(* Logix 5000 project; controller RN21_Architecture 1769-L16ER-BB1B rev 35.11; software revision 35.00; part 2 of 9 *)

ADD_ON_INSTRUCTION AOI_LOGIN_Arch   (* revision 1.0 *)
VAR_INPUT
   FBI_DataLogTrig : BOOL; {required}   // Trigger Bit for Data Log Generation
END_VAR
VAR_IN_OUT
   FBO_TriggerBit : BOOL; {required}   // Server Trigger Bit
   FBIO_Src : UDT_Login; {required}   // Source UDT Data
   FBIO_Ser : UDT_Login; {required}   // Server UDT Data
END_VAR
VAR_INPUT
   FBI_PLCServerCommFailed : BOOL; {access None, required}   // PLC to Server Communication Fail Timer Done
END_VAR
VAR_IN_OUT
   FBIO_SerUniqueNum : DINT; {required}   // Server Unique Number(Server UID)
   FBIO_SrcUniqueNum : DINT; {required}   // Source Unique Number (PLC UID)
END_VAR
VAR
   FBL_Buff : UDT_Login[100]; {access None}   // Buffer UDT Data
   FBL_Sec : UDT_Login; {access None}   // Secondary UDT Data
   FBL_IndexStore : DINT; {access None}   // Index Store Value
   FBL_Bit4 : BOOL; {access None}   // Primary Movement Completed
   FBL_TMR2 : TIMER := (PRE := 50, ACC := 1); {access None}   // Source UID Reset Delay
   FBL_Bit1 : BOOL; {access None}   // Source UID Reset
   FBL_Bit2 : BOOL; {access None}   // Source UID Less than Server UID
   FBL_Bit6 : BOOL; {access None}   // Data Moving From Secondary to Server
   FBL_TMR3 : TIMER := (PRE := 5000, ACC := 5); {access None}   // Load Movement Delay
   FBL_Bit5 : BOOL; {access None}   // Data Load From Buffer to Secondary Flag
   FBL_IndexLoad : DINT; {access None}   // Index Load Value
   FBL_Bit3 : BOOL; {access None}   // Secondary Movement Completed
   FBL_TMR1 : TIMER := (PRE := 5000); {access None}   // Server UID Movement Delay
   FBL_PrimUniqueNum : DINT; {access None}   // Primary Unique Number (PLC UID)
   FBL_BuffUniqueNum : DINT[100]; {access None}   // Buffer Unique Number (PLC UID)
   FBL_SecUniqueNum : DINT; {access None}   // Secondary Unique Number (PLC UID)
   FBL_Prim : UDT_Login; {access None}   // Primary UDT Data
   FBL_ONS : DINT; {access None}   // Common ONS DINT
   TMRDlyDatalogTrig : TIMER := (PRE := 1); {access None}
END_VAR

ROUTINE Logic   (* ladder *)
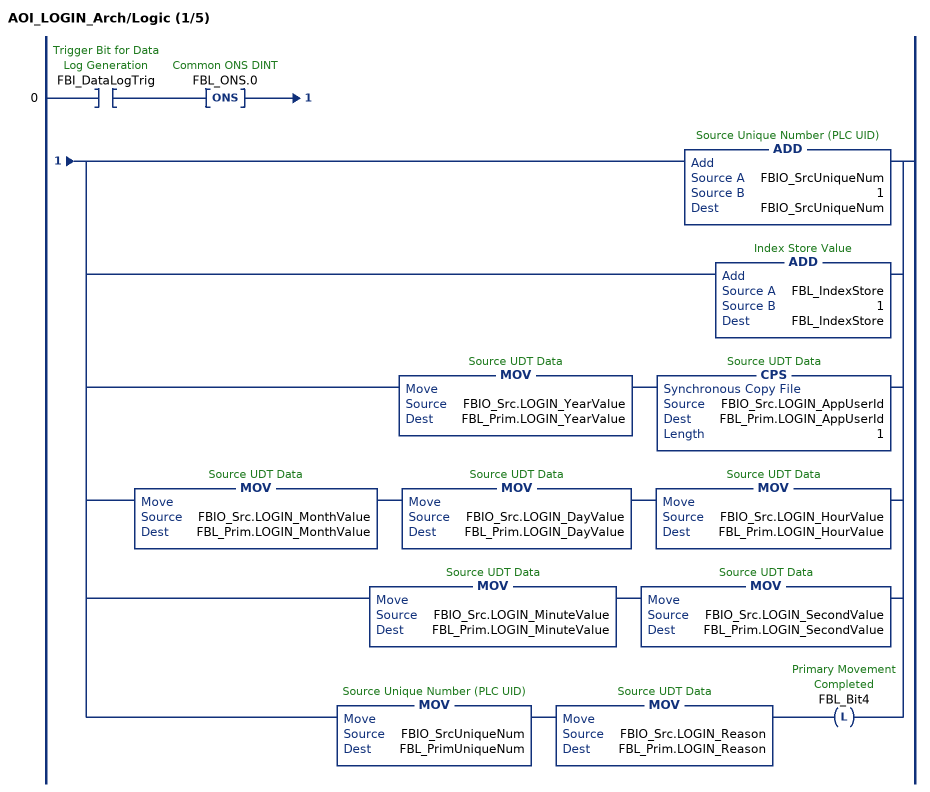
   0: XIC(FBI_DataLogTrig)ONS(FBL_ONS.0)[ADD(FBIO_SrcUniqueNum,1,FBIO_SrcUniqueNum) ,ADD(FBL_IndexStore,1,FBL_IndexStore) ,MOV(FBIO_Src.LOGIN_YearValue,FBL_Prim.LOGIN_YearValue) CPS(FBIO_Src.LOGIN_AppUserId,FBL_Prim.LOGIN_AppUserId,1) ,MOV(FBIO_Src.LOGIN_MonthValue,FBL_Prim.LOGIN_MonthValue) MOV(FBIO_Src.LOGIN_DayValue,FBL_Prim.LOGIN_DayValue) MOV(FBIO_Src.LOGIN_HourValue,FBL_Prim.LOGIN_HourValue) ,MOV(FBIO_Src.LOGIN_MinuteValue,FBL_Prim.LOGIN_MinuteValue) MOV(FBIO_Src.LOGIN_SecondValue,FBL_Prim.LOGIN_SecondValue) ,MOV(FBIO_SrcUniqueNum,FBL_PrimUniqueNum) MOV(FBIO_Src.LOGIN_Reason,FBL_Prim.LOGIN_Reason) OTL(FBL_Bit4) ];
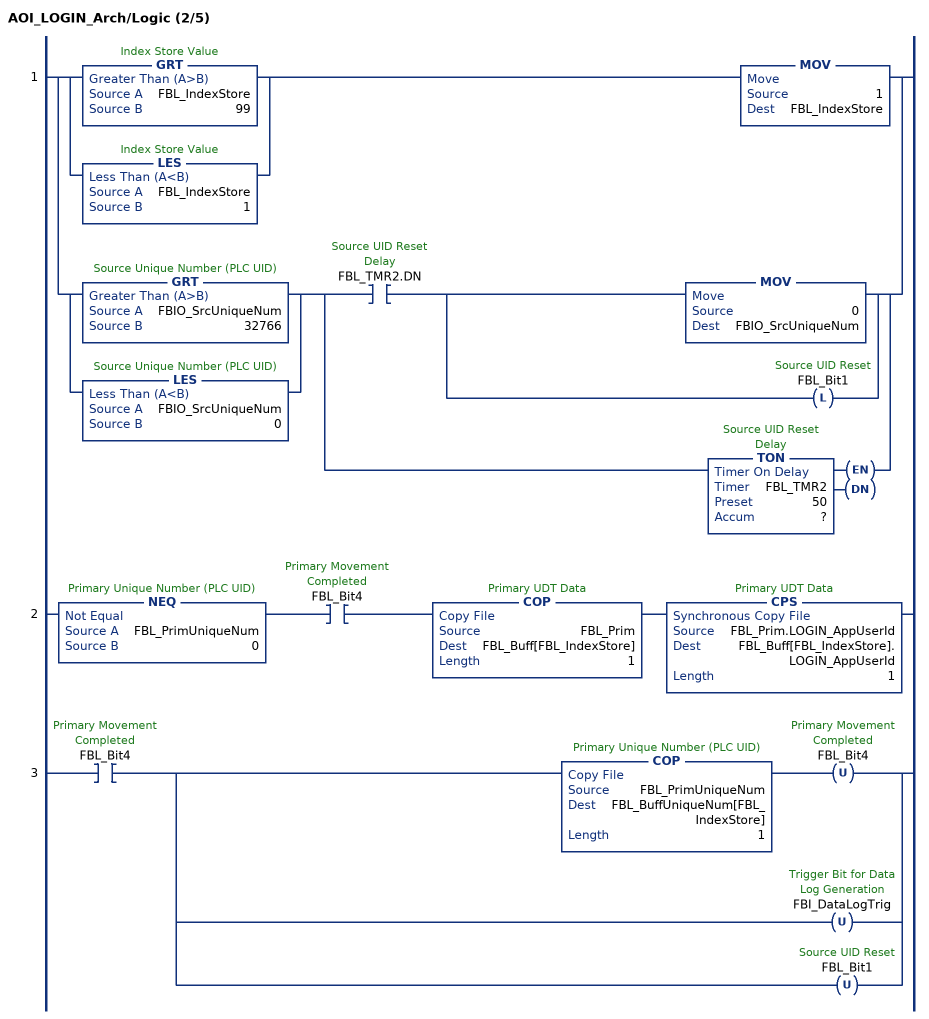
   1: [[GRT(FBL_IndexStore,99) ,LES(FBL_IndexStore,1) ] MOV(1,FBL_IndexStore) ,[GRT(FBIO_SrcUniqueNum,32766) ,LES(FBIO_SrcUniqueNum,0) ] [XIC(FBL_TMR2.DN) [MOV(0,FBIO_SrcUniqueNum) ,OTL(FBL_Bit1) ] ,TON(FBL_TMR2,?,?) ] ];
   2: NEQ(FBL_PrimUniqueNum,0)XIC(FBL_Bit4)COP(FBL_Prim,FBL_Buff[FBL_IndexStore],1)CPS(FBL_Prim.LOGIN_AppUserId,FBL_Buff[FBL_IndexStore].LOGIN_AppUserId,1);
   3: XIC(FBL_Bit4)[COP(FBL_PrimUniqueNum,FBL_BuffUniqueNum[FBL_IndexStore],1) OTU(FBL_Bit4) ,OTU(FBI_DataLogTrig) ,OTU(FBL_Bit1) ];
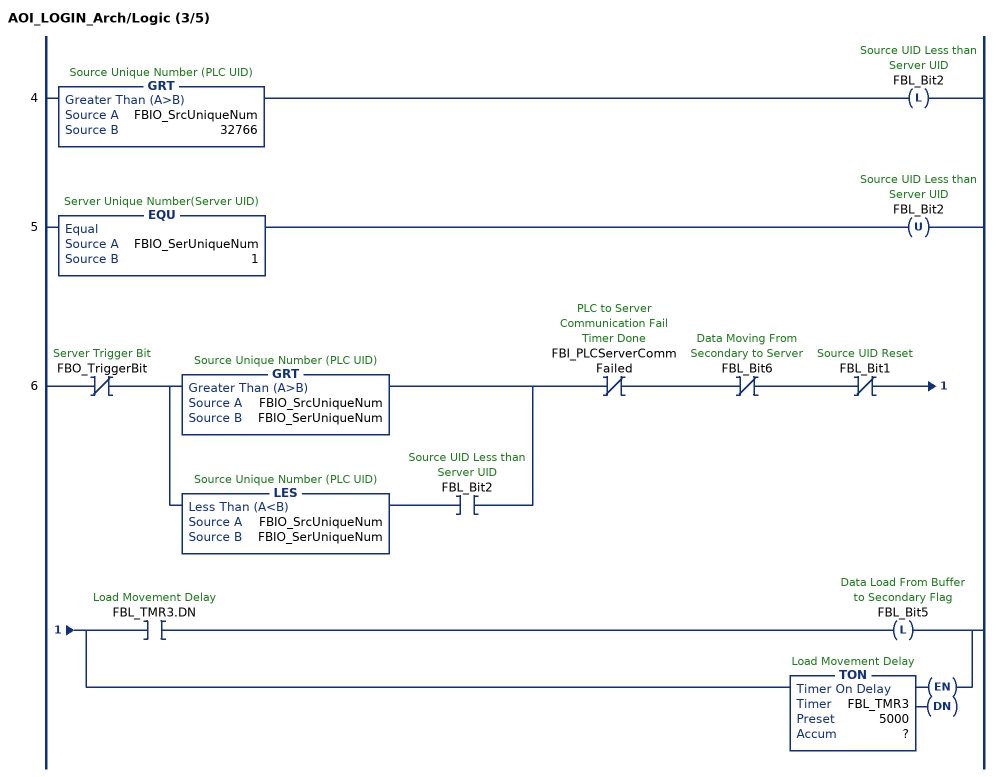
   4: GRT(FBIO_SrcUniqueNum,32766)OTL(FBL_Bit2);
   5: EQU(FBIO_SerUniqueNum,1)OTU(FBL_Bit2);
   6: XIO(FBO_TriggerBit)[GRT(FBIO_SrcUniqueNum,FBIO_SerUniqueNum) ,LES(FBIO_SrcUniqueNum,FBIO_SerUniqueNum) XIC(FBL_Bit2) ]XIO(FBI_PLCServerCommFailed)XIO(FBL_Bit6)XIO(FBL_Bit1)[XIC(FBL_TMR3.DN) OTL(FBL_Bit5) ,TON(FBL_TMR3,?,?) ];
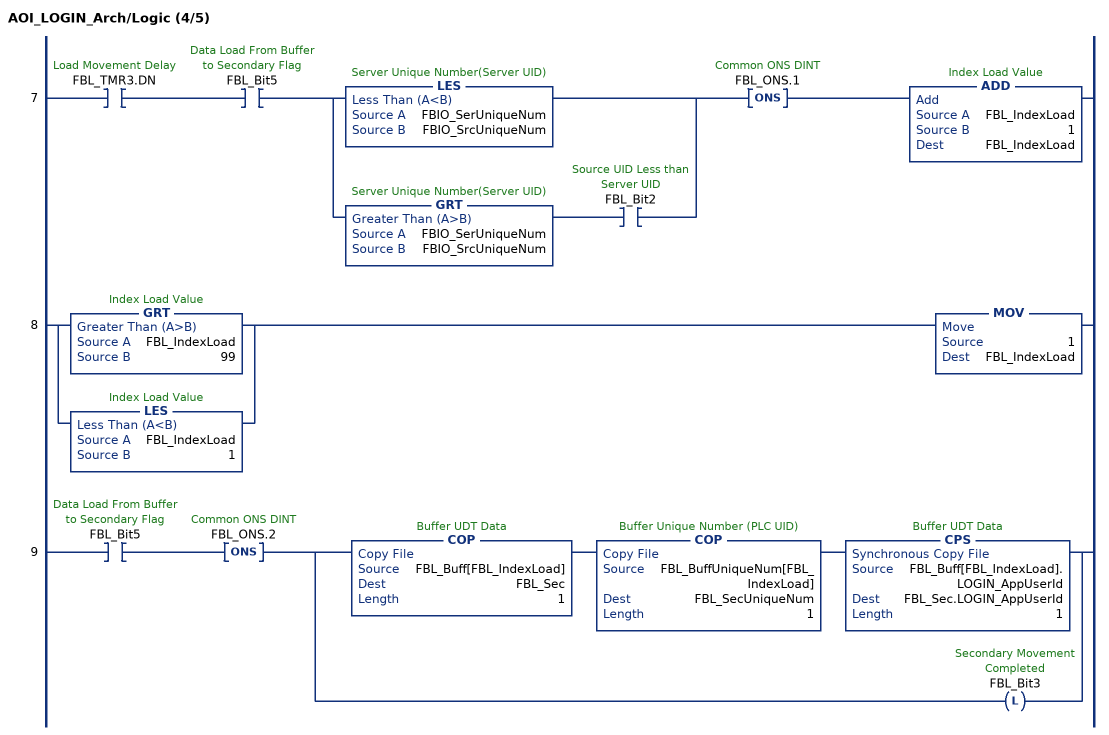
   7: XIC(FBL_TMR3.DN)XIC(FBL_Bit5)[LES(FBIO_SerUniqueNum,FBIO_SrcUniqueNum) ,GRT(FBIO_SerUniqueNum,FBIO_SrcUniqueNum) XIC(FBL_Bit2) ]ONS(FBL_ONS.1)ADD(FBL_IndexLoad,1,FBL_IndexLoad);
   8: [GRT(FBL_IndexLoad,99) ,LES(FBL_IndexLoad,1) ]MOV(1,FBL_IndexLoad);
   9: XIC(FBL_Bit5)ONS(FBL_ONS.2)[COP(FBL_Buff[FBL_IndexLoad],FBL_Sec,1) COP(FBL_BuffUniqueNum[FBL_IndexLoad],FBL_SecUniqueNum,1) CPS(FBL_Buff[FBL_IndexLoad].LOGIN_AppUserId,FBL_Sec.LOGIN_AppUserId,1) ,OTL(FBL_Bit3) ];
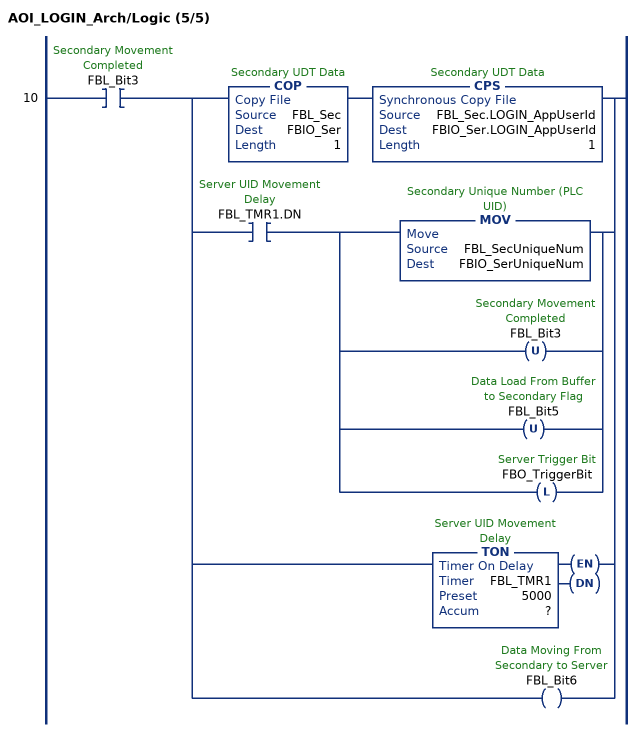
   10: XIC(FBL_Bit3)[COP(FBL_Sec,FBIO_Ser,1) CPS(FBL_Sec.LOGIN_AppUserId,FBIO_Ser.LOGIN_AppUserId,1) ,XIC(FBL_TMR1.DN) [MOV(FBL_SecUniqueNum,FBIO_SerUniqueNum) ,OTU(FBL_Bit3) ,OTU(FBL_Bit5) ,OTL(FBO_TriggerBit) ] ,TON(FBL_TMR1,?,?) ,OTE(FBL_Bit6) ];
END_ROUTINE
END_ADD_ON_INSTRUCTION

ADD_ON_INSTRUCTION AOI_PDL_Arch   (* revision 1.0 *)
VAR_INPUT
   FBI_DataLogTrig : BOOL; {required}   // Trigger Bit for Data Log Generation
END_VAR
VAR_IN_OUT
   FBO_TriggerBit : BOOL; {required}   // Server Trigger Bit
   FBIO_Src : UDT_Process; {required}   // Source UDT Data
   FBIO_Ser : UDT_Process; {required}   // Server UDT Data
END_VAR
VAR_INPUT
   FBI_PLCServerCommFailed : BOOL; {access None, required}   // PLC to Server Communication Fail Timer Done
END_VAR
VAR_IN_OUT
   FBIO_SerUniqueNum : DINT; {required}   // Server Unique Number(Server UID)
   FBIO_SrcUniqueNum : DINT; {required}   // Source Unique Number (PLC UID)
END_VAR
VAR
   FBL_Prim : UDT_Process; {access None}   // Primary UDT Data
   FBL_Buff : UDT_Process[100]; {access None}   // Buffer UDT Data
   FBL_Sec : UDT_Process; {access None}   // Secondary UDT Data
   FBL_IndexStore : DINT; {access None}   // Index Store Value
   FBL_Bit4 : BOOL; {access None}   // Primary Movement Completed
   FBL_TMR2 : TIMER := (PRE := 1, ACC := 1); {access None}   // Source UID Reset Delay
   FBL_Bit1 : BOOL; {access None}   // Source UID Reset
   FBL_Bit2 : BOOL; {access None}   // Source UID Less than Server UID
   FBL_Bit6 : BOOL; {access None}   // Data Moving From Secondary to Server
   FBL_TMR3 : TIMER := (PRE := 5000, ACC := 5); {access None}   // Load Movement Delay
   FBL_Bit5 : BOOL; {access None}   // Data Load From Buffer to Secondary Flag
   FBL_IndexLoad : DINT; {access None}   // Index Load Value
   FBL_Bit3 : BOOL; {access None}   // Secondary Movement Completed
   FBL_TMR1 : TIMER := (PRE := 5000); {access None}   // Server UID Movement Delay
   FBL_PrimUniqueNum : DINT; {access None}   // Primary Unique Number (PLC UID)
   FBL_BuffUniqueNum : DINT[100]; {access None}   // Buffer Unique Number (PLC UID)
   FBL_SecUniqueNum : DINT; {access None}   // Secondary Unique Number (PLC UID)
   FBL_ONS : DINT; {access None}   // Common ONS DINT
END_VAR

ROUTINE Logic   (* ladder *)
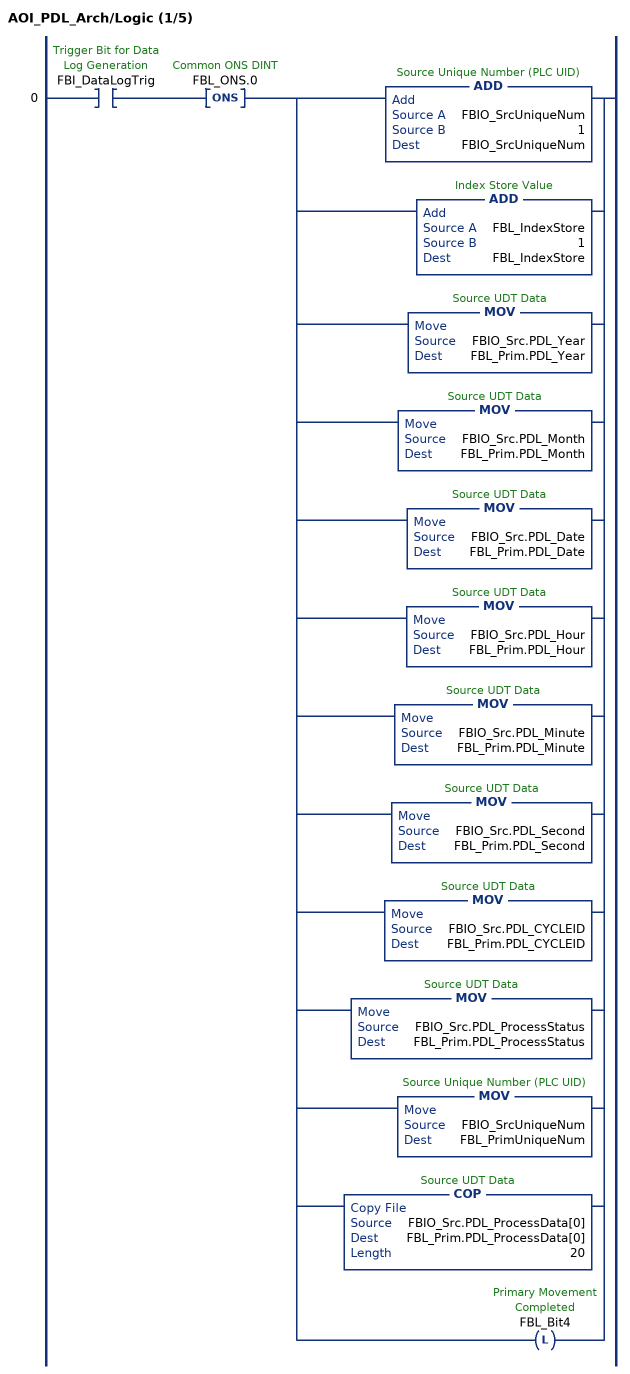
   0: XIC(FBI_DataLogTrig)ONS(FBL_ONS.0)[ADD(FBIO_SrcUniqueNum,1,FBIO_SrcUniqueNum) ,ADD(FBL_IndexStore,1,FBL_IndexStore) ,MOV(FBIO_Src.PDL_Year,FBL_Prim.PDL_Year) ,MOV(FBIO_Src.PDL_Month,FBL_Prim.PDL_Month) ,MOV(FBIO_Src.PDL_Date,FBL_Prim.PDL_Date) ,MOV(FBIO_Src.PDL_Hour,FBL_Prim.PDL_Hour) ,MOV(FBIO_Src.PDL_Minute,FBL_Prim.PDL_Minute) ,MOV(FBIO_Src.PDL_Second,FBL_Prim.PDL_Second) ,MOV(FBIO_Src.PDL_CYCLEID,FBL_Prim.PDL_CYCLEID) ,MOV(FBIO_Src.PDL_ProcessStatus,FBL_Prim.PDL_ProcessStatus) ,MOV(FBIO_SrcUniqueNum,FBL_PrimUniqueNum) ,COP(FBIO_Src.PDL_ProcessData[0],FBL_Prim.PDL_ProcessData[0],20) ,OTL(FBL_Bit4) ];
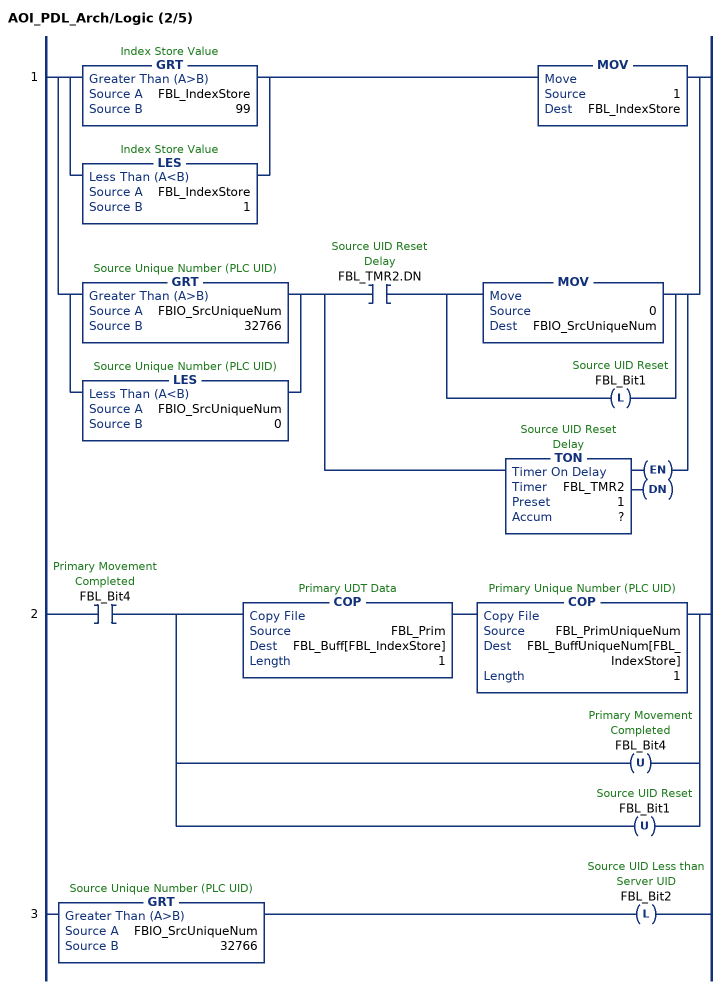
   1: [[GRT(FBL_IndexStore,99) ,LES(FBL_IndexStore,1) ] MOV(1,FBL_IndexStore) ,[GRT(FBIO_SrcUniqueNum,32766) ,LES(FBIO_SrcUniqueNum,0) ] [XIC(FBL_TMR2.DN) [MOV(0,FBIO_SrcUniqueNum) ,OTL(FBL_Bit1) ] ,TON(FBL_TMR2,?,?) ] ];
   2: XIC(FBL_Bit4)[COP(FBL_Prim,FBL_Buff[FBL_IndexStore],1) COP(FBL_PrimUniqueNum,FBL_BuffUniqueNum[FBL_IndexStore],1) ,OTU(FBL_Bit4) ,OTU(FBL_Bit1) ];
   3: GRT(FBIO_SrcUniqueNum,32766)OTL(FBL_Bit2);
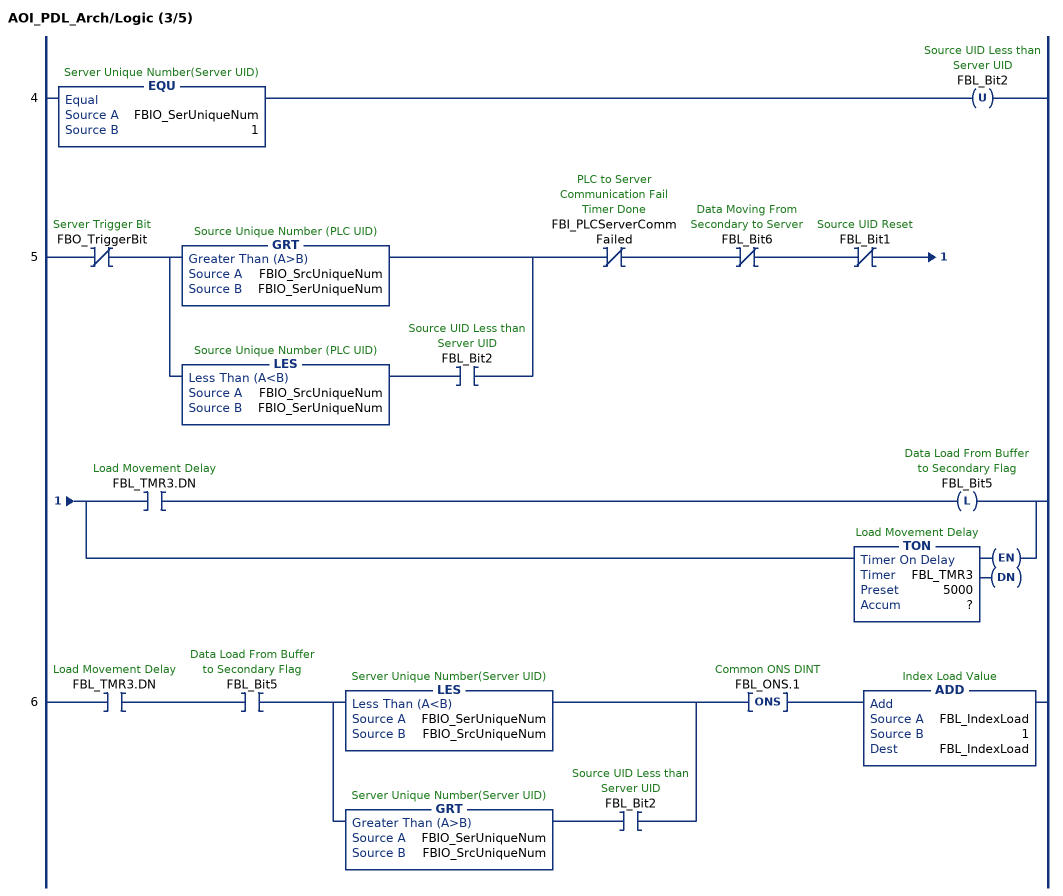
   4: EQU(FBIO_SerUniqueNum,1)OTU(FBL_Bit2);
   5: XIO(FBO_TriggerBit)[GRT(FBIO_SrcUniqueNum,FBIO_SerUniqueNum) ,LES(FBIO_SrcUniqueNum,FBIO_SerUniqueNum) XIC(FBL_Bit2) ]XIO(FBI_PLCServerCommFailed)XIO(FBL_Bit6)XIO(FBL_Bit1)[XIC(FBL_TMR3.DN) OTL(FBL_Bit5) ,TON(FBL_TMR3,?,?) ];
   6: XIC(FBL_TMR3.DN)XIC(FBL_Bit5)[LES(FBIO_SerUniqueNum,FBIO_SrcUniqueNum) ,GRT(FBIO_SerUniqueNum,FBIO_SrcUniqueNum) XIC(FBL_Bit2) ]ONS(FBL_ONS.1)ADD(FBL_IndexLoad,1,FBL_IndexLoad);
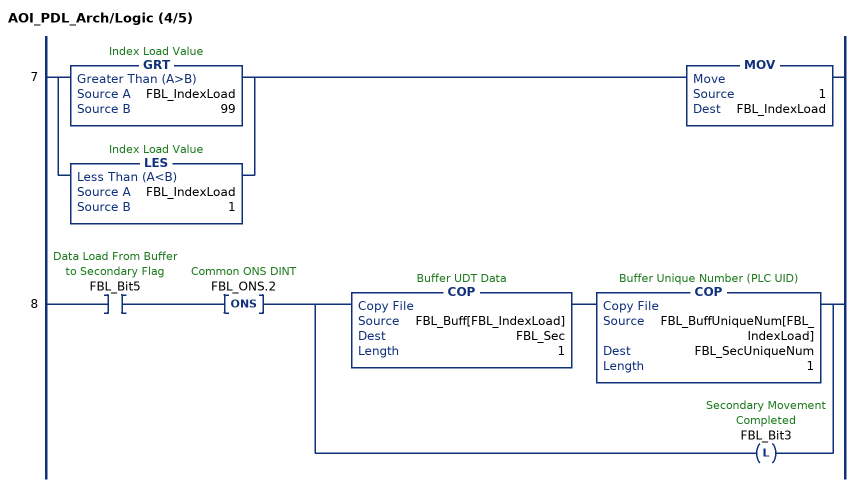
   7: [GRT(FBL_IndexLoad,99) ,LES(FBL_IndexLoad,1) ]MOV(1,FBL_IndexLoad);
   8: XIC(FBL_Bit5)ONS(FBL_ONS.2)[COP(FBL_Buff[FBL_IndexLoad],FBL_Sec,1) COP(FBL_BuffUniqueNum[FBL_IndexLoad],FBL_SecUniqueNum,1) ,OTL(FBL_Bit3) ];
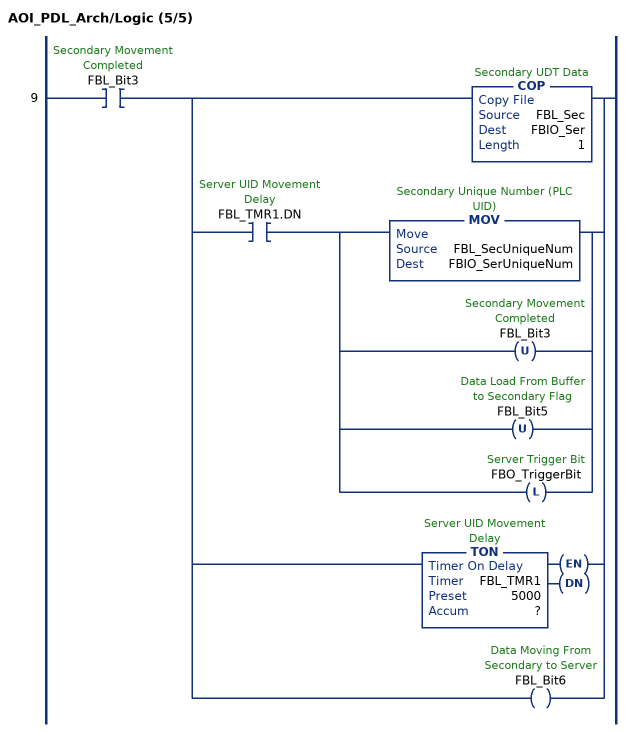
   9: XIC(FBL_Bit3)[COP(FBL_Sec,FBIO_Ser,1) ,XIC(FBL_TMR1.DN) [MOV(FBL_SecUniqueNum,FBIO_SerUniqueNum) ,OTU(FBL_Bit3) ,OTU(FBL_Bit5) ,OTL(FBO_TriggerBit) ] ,TON(FBL_TMR1,?,?) ,OTE(FBL_Bit6) ];
END_ROUTINE
END_ADD_ON_INSTRUCTION

ADD_ON_INSTRUCTION AOI_PDL_DataCapture   (* revision 1.0 *)
VAR_INPUT
   FBI_IsPrintIntervalReq : BOOL; {required}
   FBI_PrintInterval : INT; {required}
END_VAR
VAR_OUTPUT
   FBO_RUNNINGSTSMOVTRIG : BOOL; {access Read Only, required}
END_VAR
VAR_INPUT
   FBI_STOP : BOOL; {required}
   FBI_START : BOOL; {required}
END_VAR
VAR_OUTPUT
   FBO_STARTED : BOOL; {required}
END_VAR
VAR_INPUT
   FBI_PAUSE_RELEASE : BOOL; {required}
   FBI_OneSecTrig : BOOL; {required}
   FBI_COMPLETED : BOOL; {required}
   FBI_ALARM : BOOL; {required}
END_VAR
VAR_OUTPUT
   FBO_STOPEDSTSMOVTRIG : BOOL; {required}
   FBO_PAUSEDSTSMOVTRIG : BOOL; {required}
   FBO_STOPEDALARMSTSMOVTRIG : BOOL; {required}
   FBO_RELEASEDSTSMOVTRIG : BOOL; {required}
END_VAR
VAR_INPUT
   FBIPROCESSRESET : BOOL; {required}
END_VAR
VAR_OUTPUT
   FBO_CMPLTSTSMOVTRIG : BOOL; {access None, required}
END_VAR
VAR_INPUT
   FBI_Enable : BOOL; {required}
END_VAR
VAR_OUTPUT
   FBO_Active : BOOL; {required}
END_VAR
VAR_INPUT
   FBIO_AlarmReset : BOOL; {required}
END_VAR
VAR_OUTPUT
   FBO_PAUSED : BOOL; {access None, required}
   FBO_FAULT : BOOL; {access None}
END_VAR
VAR
   CTU_PrintInterval : COUNTER; {access None}
   FBL_Bit1 : BOOL; {access None}
   FBL_Bit2 : BOOL; {access None}
   FBL_Bit3 : BOOL; {access None}
   TMR_CycleTrigDly : TIMER := (PRE := 200); {access None}
   FBL_ReleaseReq : BOOL; {access None}
   FBL_StartReqFlag : BOOL; {access None}
   FBL_StartLatch : BOOL; {access None}
   ONS : DINT; {access None}
   TMR_ResetDly1 : TIMER := (PRE := 1000); {access None}
   FBL_ReleaseReqFlag : BOOL; {access None}
   FBL_RunningFlag : BOOL; {access None}
   TMR_RunTrigDly : TIMER := (PRE := 400); {access None}
   FBL_StartReqFlag1 : BOOL; {access None}
   FBL_Pause_Req : BOOL; {access None}
   FBL_ReleaseReqFlag1 : BOOL; {access None}
END_VAR

ROUTINE Logic   (* ladder *)
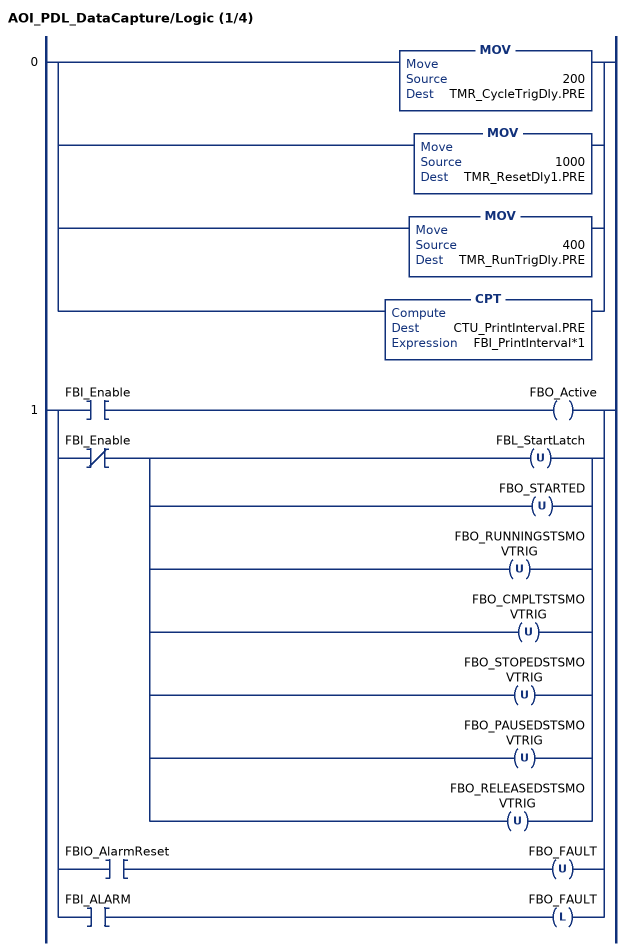
   0: [MOV(200,TMR_CycleTrigDly.PRE) ,MOV(1000,TMR_ResetDly1.PRE) ,MOV(400,TMR_RunTrigDly.PRE) ,CPT(CTU_PrintInterval.PRE,FBI_PrintInterval*1) ];
   1: [XIC(FBI_Enable) OTE(FBO_Active) ,XIO(FBI_Enable) [OTU(FBL_StartLatch) ,OTU(FBO_STARTED) ,OTU(FBO_RUNNINGSTSMOVTRIG) ,OTU(FBO_CMPLTSTSMOVTRIG) ,OTU(FBO_STOPEDSTSMOVTRIG) ,OTU(FBO_PAUSEDSTSMOVTRIG) ,OTU(FBO_RELEASEDSTSMOVTRIG) ] ,XIC(FBIO_AlarmReset) OTU(FBO_FAULT) ,XIC(FBI_ALARM) OTL(FBO_FAULT) ];
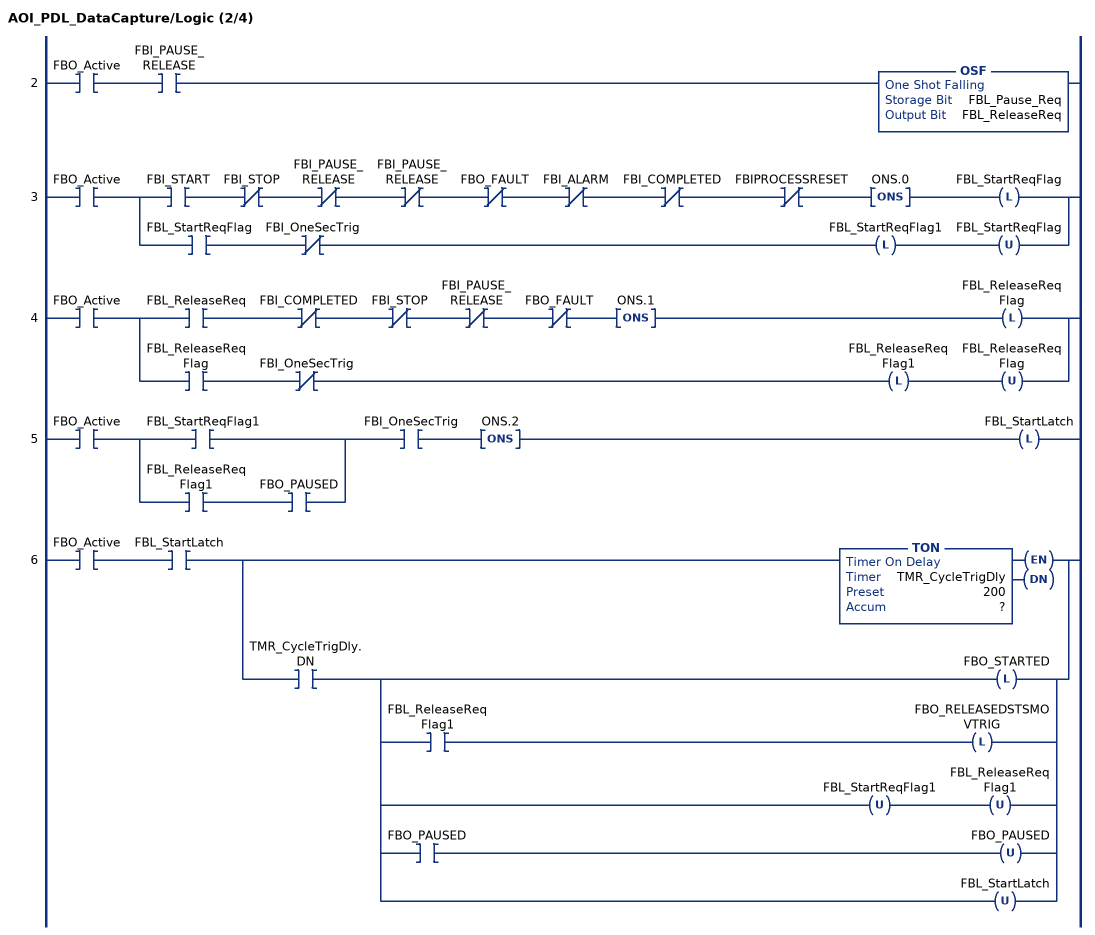
   2: XIC(FBO_Active)XIC(FBI_PAUSE_RELEASE)OSF(FBL_Pause_Req,FBL_ReleaseReq);
   3: XIC(FBO_Active)[XIC(FBI_START) XIO(FBI_STOP) XIO(FBI_PAUSE_RELEASE) XIO(FBI_PAUSE_RELEASE) XIO(FBO_FAULT) XIO(FBI_ALARM) XIO(FBI_COMPLETED) XIO(FBIPROCESSRESET) ONS(ONS.0) OTL(FBL_StartReqFlag) ,XIC(FBL_StartReqFlag) XIO(FBI_OneSecTrig) OTL(FBL_StartReqFlag1) OTU(FBL_StartReqFlag) ];
   4: XIC(FBO_Active)[XIC(FBL_ReleaseReq) XIO(FBI_COMPLETED) XIO(FBI_STOP) XIO(FBI_PAUSE_RELEASE) XIO(FBO_FAULT) ONS(ONS.1) OTL(FBL_ReleaseReqFlag) ,XIC(FBL_ReleaseReqFlag) XIO(FBI_OneSecTrig) OTL(FBL_ReleaseReqFlag1) OTU(FBL_ReleaseReqFlag) ];
   5: XIC(FBO_Active)[XIC(FBL_StartReqFlag1) ,XIC(FBL_ReleaseReqFlag1) XIC(FBO_PAUSED) ]XIC(FBI_OneSecTrig)ONS(ONS.2)OTL(FBL_StartLatch);
   6: XIC(FBO_Active)XIC(FBL_StartLatch)[TON(TMR_CycleTrigDly,?,?) ,XIC(TMR_CycleTrigDly.DN) [OTL(FBO_STARTED) ,XIC(FBL_ReleaseReqFlag1) OTL(FBO_RELEASEDSTSMOVTRIG) ,OTU(FBL_StartReqFlag1) OTU(FBL_ReleaseReqFlag1) ,XIC(FBO_PAUSED) OTU(FBO_PAUSED) ,OTU(FBL_StartLatch) ] ];
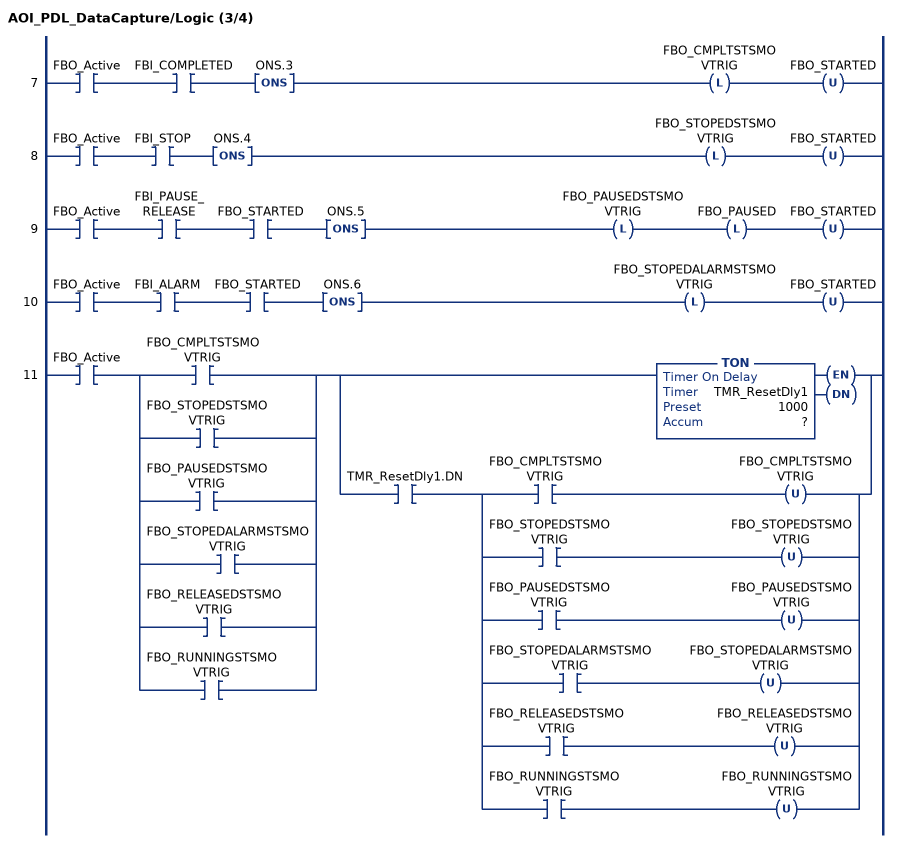
   7: XIC(FBO_Active)XIC(FBI_COMPLETED)ONS(ONS.3)OTL(FBO_CMPLTSTSMOVTRIG)OTU(FBO_STARTED);
   8: XIC(FBO_Active)XIC(FBI_STOP)ONS(ONS.4)OTL(FBO_STOPEDSTSMOVTRIG)OTU(FBO_STARTED);
   9: XIC(FBO_Active)XIC(FBI_PAUSE_RELEASE)XIC(FBO_STARTED)ONS(ONS.5)OTL(FBO_PAUSEDSTSMOVTRIG)OTL(FBO_PAUSED)OTU(FBO_STARTED);
   10: XIC(FBO_Active)XIC(FBI_ALARM)XIC(FBO_STARTED)ONS(ONS.6)OTL(FBO_STOPEDALARMSTSMOVTRIG)OTU(FBO_STARTED);
   11: XIC(FBO_Active)[XIC(FBO_CMPLTSTSMOVTRIG) ,XIC(FBO_STOPEDSTSMOVTRIG) ,XIC(FBO_PAUSEDSTSMOVTRIG) ,XIC(FBO_STOPEDALARMSTSMOVTRIG) ,XIC(FBO_RELEASEDSTSMOVTRIG) ,XIC(FBO_RUNNINGSTSMOVTRIG) ][TON(TMR_ResetDly1,?,?) ,XIC(TMR_ResetDly1.DN) [XIC(FBO_CMPLTSTSMOVTRIG) OTU(FBO_CMPLTSTSMOVTRIG) ,XIC(FBO_STOPEDSTSMOVTRIG) OTU(FBO_STOPEDSTSMOVTRIG) ,XIC(FBO_PAUSEDSTSMOVTRIG) OTU(FBO_PAUSEDSTSMOVTRIG) ,XIC(FBO_STOPEDALARMSTSMOVTRIG) OTU(FBO_STOPEDALARMSTSMOVTRIG) ,XIC(FBO_RELEASEDSTSMOVTRIG) OTU(FBO_RELEASEDSTSMOVTRIG) ,XIC(FBO_RUNNINGSTSMOVTRIG) OTU(FBO_RUNNINGSTSMOVTRIG) ] ];
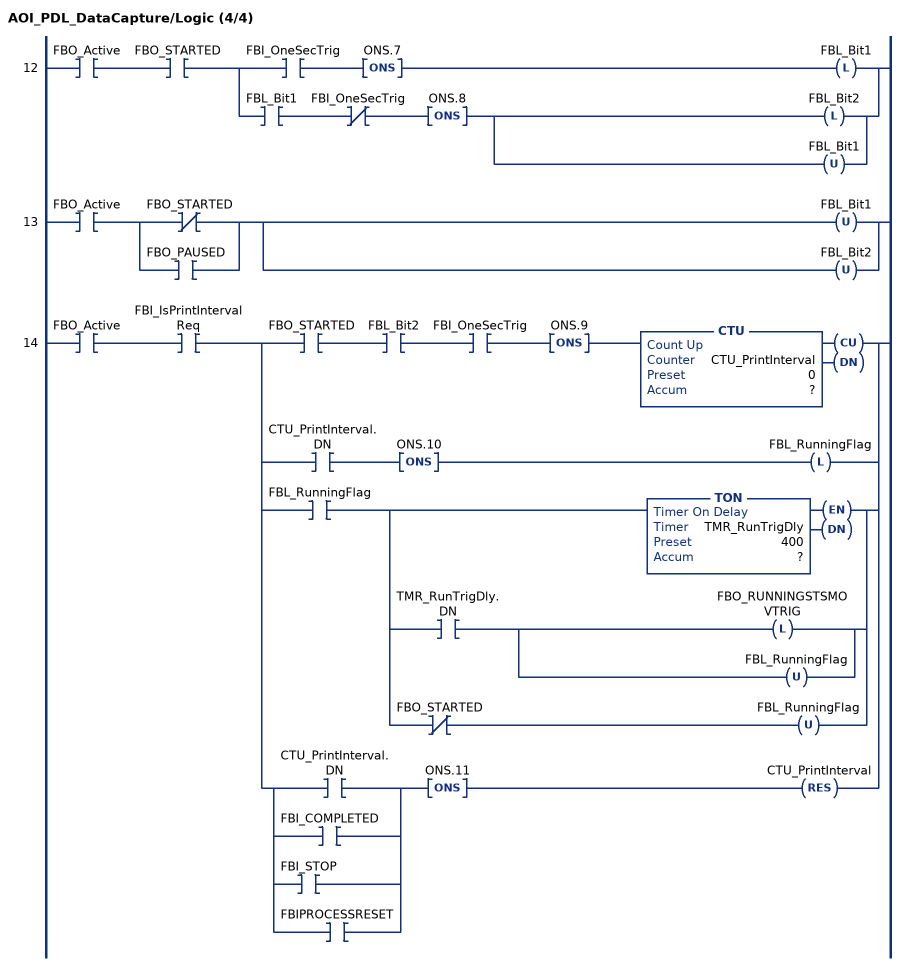
   12: XIC(FBO_Active)XIC(FBO_STARTED)[XIC(FBI_OneSecTrig) ONS(ONS.7) OTL(FBL_Bit1) ,XIC(FBL_Bit1) XIO(FBI_OneSecTrig) ONS(ONS.8) [OTL(FBL_Bit2) ,OTU(FBL_Bit1) ] ];
   13: XIC(FBO_Active)[XIO(FBO_STARTED) ,XIC(FBO_PAUSED) ][OTU(FBL_Bit1) ,OTU(FBL_Bit2) ];
   14: XIC(FBO_Active)XIC(FBI_IsPrintIntervalReq)[XIC(FBO_STARTED) XIC(FBL_Bit2) XIC(FBI_OneSecTrig) ONS(ONS.9) CTU(CTU_PrintInterval,?,?) ,XIC(CTU_PrintInterval.DN) ONS(ONS.10) OTL(FBL_RunningFlag) ,XIC(FBL_RunningFlag) [TON(TMR_RunTrigDly,?,?) ,XIC(TMR_RunTrigDly.DN) [OTL(FBO_RUNNINGSTSMOVTRIG) ,OTU(FBL_RunningFlag) ] ,XIO(FBO_STARTED) OTU(FBL_RunningFlag) ] ,[XIC(CTU_PrintInterval.DN) ,XIC(FBI_COMPLETED) ,XIC(FBI_STOP) ,XIC(FBIPROCESSRESET) ] ONS(ONS.11) RES(CTU_PrintInterval) ];
END_ROUTINE
END_ADD_ON_INSTRUCTION

ADD_ON_INSTRUCTION AOI_RP_Arch   (* revision 1.0 *)
VAR_INPUT
   FBI_DataLogTrig : BOOL; {required}   // Trigger Bit for Data Log Generation
END_VAR
VAR_IN_OUT
   FBO_TriggerBit : BOOL; {required}   // Server Trigger Bit
   FBIO_Src : UDT_Recipe; {required}   // Source UDT Data
   FBIO_Ser : UDT_Recipe; {required}   // Server UDT Data
END_VAR
VAR_INPUT
   FBI_PLCServerCommFailed : BOOL; {access None, required}   // PLC to Server Communication Fail Timer Done
END_VAR
VAR_IN_OUT
   FBIO_SrcUniqueNum : DINT; {required}   // Source Unique Number (PLC UID)
   FBIO_SerUniqueNum : DINT; {required}   // Server Unique Number(Server UID)
END_VAR
VAR
   FBL_Prim : UDT_Recipe; {access None}   // Primary UDT Data
   FBL_Buff : UDT_Recipe[5]; {access None}   // Buffer UDT Data
   FBL_Sec : UDT_Recipe; {access None}   // Secondary UDT Data
   FBL_IndexStore : DINT; {access None}   // Index Store Value
   FBL_Bit4 : BOOL; {access None}   // Primary Movement Completed
   FBL_TMR2 : TIMER := (PRE := 1, ACC := 1); {access None}   // Source UID Reset Delay
   FBL_Bit1 : BOOL; {access None}   // Source UID Reset
   FBL_Bit2 : BOOL; {access None}   // Source UID Less than Server UID
   FBL_Bit6 : BOOL; {access None}   // Data Moving From Secondary to Server
   FBL_TMR3 : TIMER := (PRE := 5000, ACC := 5); {access None}   // Load Movement Delay
   FBL_Bit5 : BOOL; {access None}   // Data Load From Buffer to Secondary Flag
   FBL_IndexLoad : DINT; {access None}   // Index Load Value
   FBL_Bit3 : BOOL; {access None}   // Secondary Movement Completed
   FBL_TMR1 : TIMER := (PRE := 5000); {access None}   // Server UID Movement Delay
   FBL_PrimUniqueNum : DINT; {access None}   // Primary Unique Number (PLC UID)
   FBL_BuffUniqueNum : DINT[5]; {access None}   // Buffer Unique Number (PLC UID)
   FBL_SecUniqueNum : DINT; {access None}   // Secondary Unique Number (PLC UID)
   FBL_ONS : DINT; {access None}   // Common ONS DINT
END_VAR

ROUTINE Logic   (* ladder *)
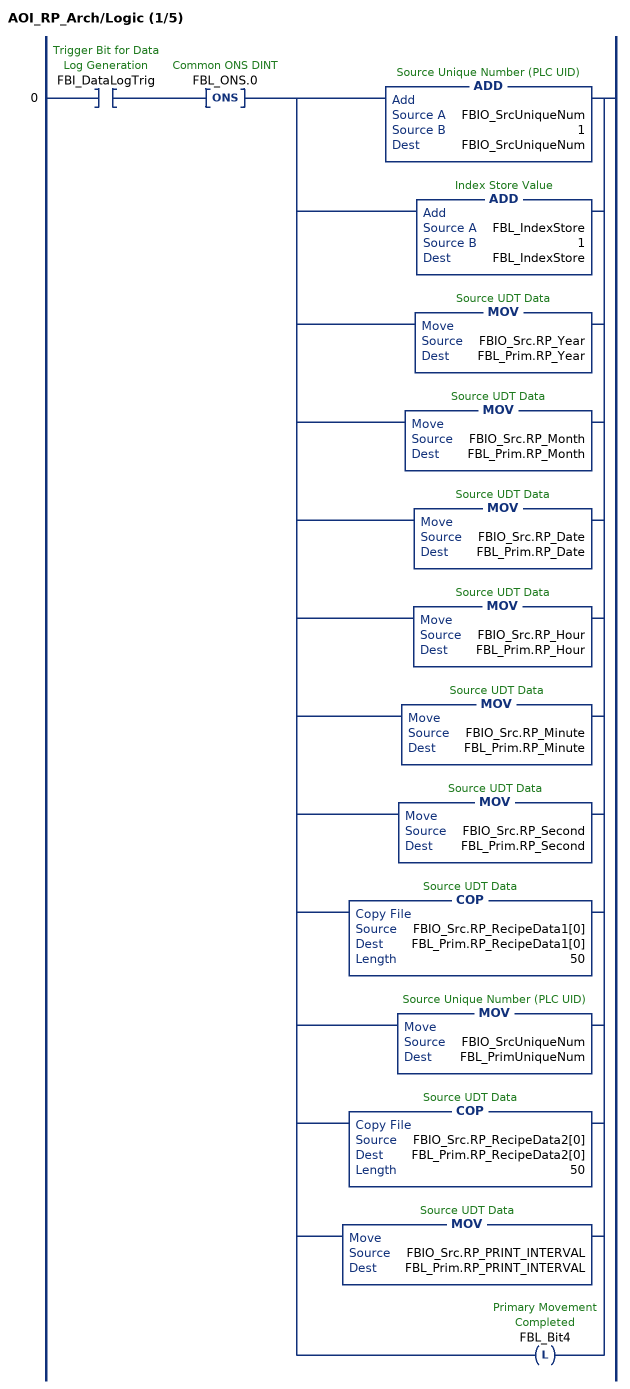
   0: XIC(FBI_DataLogTrig)ONS(FBL_ONS.0)[ADD(FBIO_SrcUniqueNum,1,FBIO_SrcUniqueNum) ,ADD(FBL_IndexStore,1,FBL_IndexStore) ,MOV(FBIO_Src.RP_Year,FBL_Prim.RP_Year) ,MOV(FBIO_Src.RP_Month,FBL_Prim.RP_Month) ,MOV(FBIO_Src.RP_Date,FBL_Prim.RP_Date) ,MOV(FBIO_Src.RP_Hour,FBL_Prim.RP_Hour) ,MOV(FBIO_Src.RP_Minute,FBL_Prim.RP_Minute) ,MOV(FBIO_Src.RP_Second,FBL_Prim.RP_Second) ,COP(FBIO_Src.RP_RecipeData1[0],FBL_Prim.RP_RecipeData1[0],50) ,MOV(FBIO_SrcUniqueNum,FBL_PrimUniqueNum) ,COP(FBIO_Src.RP_RecipeData2[0],FBL_Prim.RP_RecipeData2[0],50) ,MOV(FBIO_Src.RP_PRINT_INTERVAL,FBL_Prim.RP_PRINT_INTERVAL) ,OTL(FBL_Bit4) ];
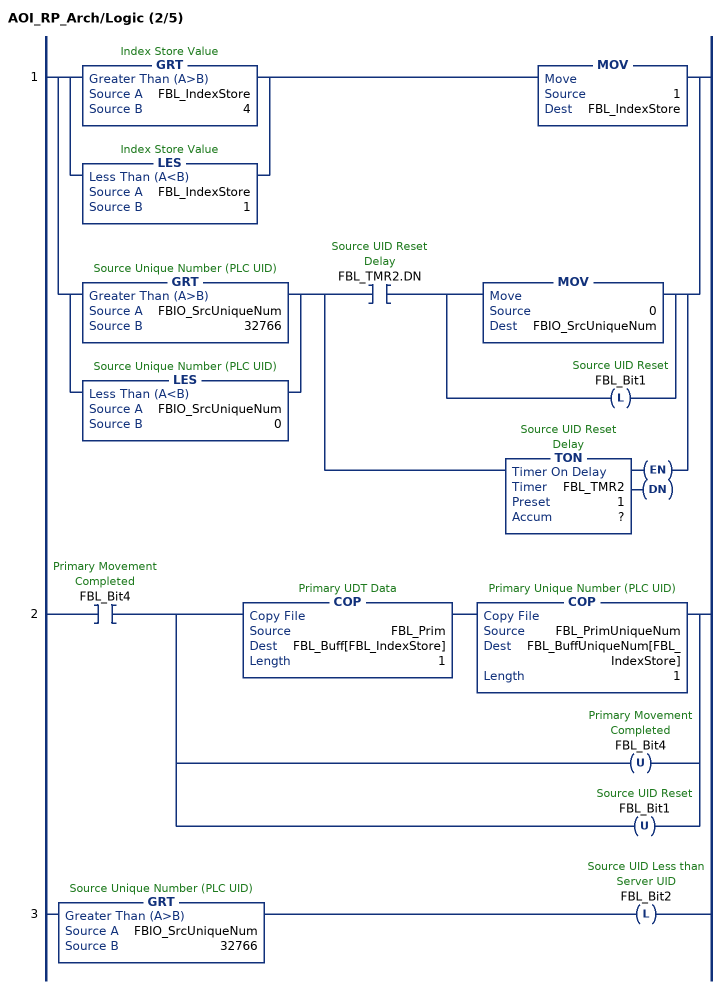
   1: [[GRT(FBL_IndexStore,4) ,LES(FBL_IndexStore,1) ] MOV(1,FBL_IndexStore) ,[GRT(FBIO_SrcUniqueNum,32766) ,LES(FBIO_SrcUniqueNum,0) ] [XIC(FBL_TMR2.DN) [MOV(0,FBIO_SrcUniqueNum) ,OTL(FBL_Bit1) ] ,TON(FBL_TMR2,?,?) ] ];
   2: XIC(FBL_Bit4)[COP(FBL_Prim,FBL_Buff[FBL_IndexStore],1) COP(FBL_PrimUniqueNum,FBL_BuffUniqueNum[FBL_IndexStore],1) ,OTU(FBL_Bit4) ,OTU(FBL_Bit1) ];
   3: GRT(FBIO_SrcUniqueNum,32766)OTL(FBL_Bit2);
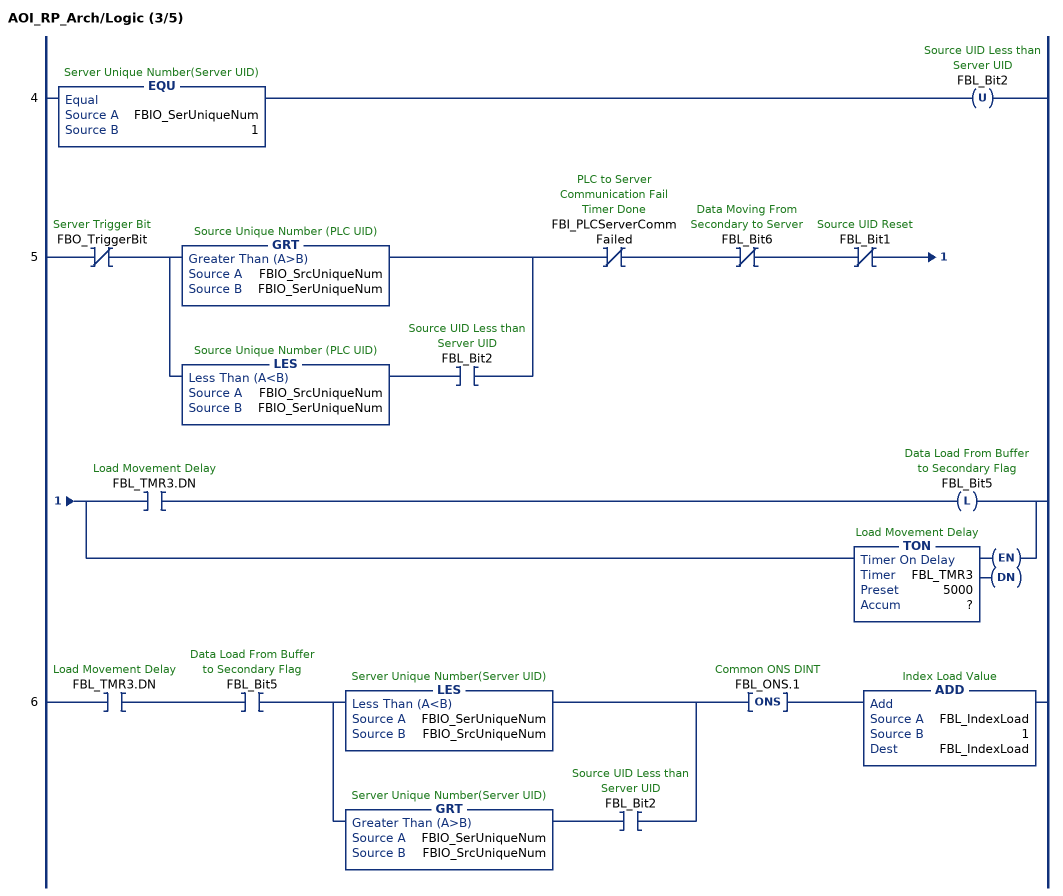
   4: EQU(FBIO_SerUniqueNum,1)OTU(FBL_Bit2);
   5: XIO(FBO_TriggerBit)[GRT(FBIO_SrcUniqueNum,FBIO_SerUniqueNum) ,LES(FBIO_SrcUniqueNum,FBIO_SerUniqueNum) XIC(FBL_Bit2) ]XIO(FBI_PLCServerCommFailed)XIO(FBL_Bit6)XIO(FBL_Bit1)[XIC(FBL_TMR3.DN) OTL(FBL_Bit5) ,TON(FBL_TMR3,?,?) ];
   6: XIC(FBL_TMR3.DN)XIC(FBL_Bit5)[LES(FBIO_SerUniqueNum,FBIO_SrcUniqueNum) ,GRT(FBIO_SerUniqueNum,FBIO_SrcUniqueNum) XIC(FBL_Bit2) ]ONS(FBL_ONS.1)ADD(FBL_IndexLoad,1,FBL_IndexLoad);
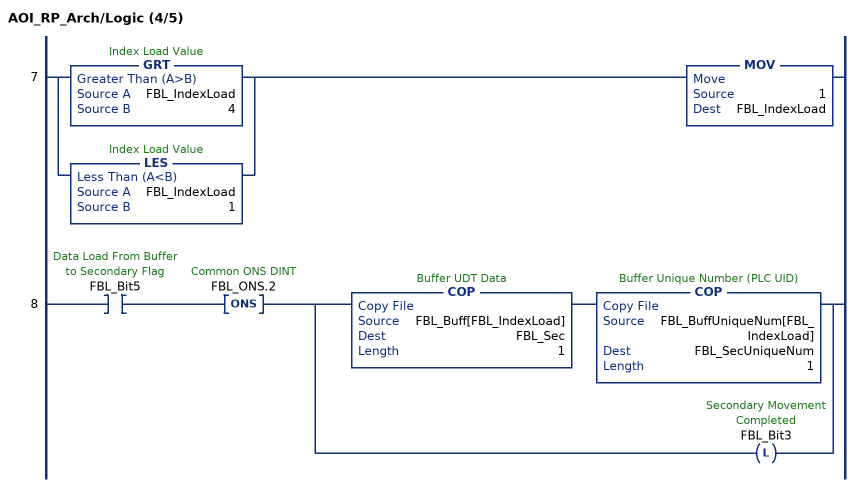
   7: [GRT(FBL_IndexLoad,4) ,LES(FBL_IndexLoad,1) ]MOV(1,FBL_IndexLoad);
   8: XIC(FBL_Bit5)ONS(FBL_ONS.2)[COP(FBL_Buff[FBL_IndexLoad],FBL_Sec,1) COP(FBL_BuffUniqueNum[FBL_IndexLoad],FBL_SecUniqueNum,1) ,OTL(FBL_Bit3) ];
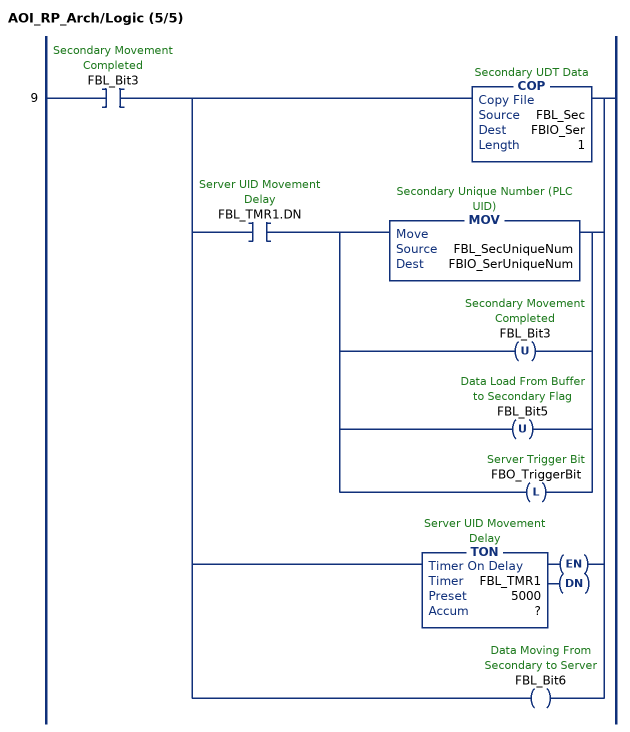
   9: XIC(FBL_Bit3)[COP(FBL_Sec,FBIO_Ser,1) ,XIC(FBL_TMR1.DN) [MOV(FBL_SecUniqueNum,FBIO_SerUniqueNum) ,OTU(FBL_Bit3) ,OTU(FBL_Bit5) ,OTL(FBO_TriggerBit) ] ,TON(FBL_TMR1,?,?) ,OTE(FBL_Bit6) ];
END_ROUTINE
END_ADD_ON_INSTRUCTION
